FUNCTION_BLOCK TwoStateCtrl (* Template for a simple Basic Function Block Type *)
  (* Standard: 61499-2 *)
  (* Version 0.0, 2016-05-26, 4DIAC-IDE, 4DIAC *)
  (* Version 1.0, 2016-05-26, AZ, 4DIAC *)
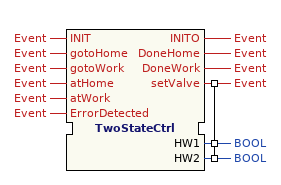
  EVENT_INPUT
    INIT; (* Initialization Request *)
    gotoHome;
    gotoWork;
    atHome;
    atWork;
    ErrorDetected;
  END_EVENT
  EVENT_OUTPUT
    INITO; (* Initialization Confirm *)
    DoneHome;
    DoneWork;
    setValve WITH HW1, HW2;
  END_EVENT
  VAR_OUTPUT
    HW1 : BOOL;
    HW2 : BOOL;
  END_VAR
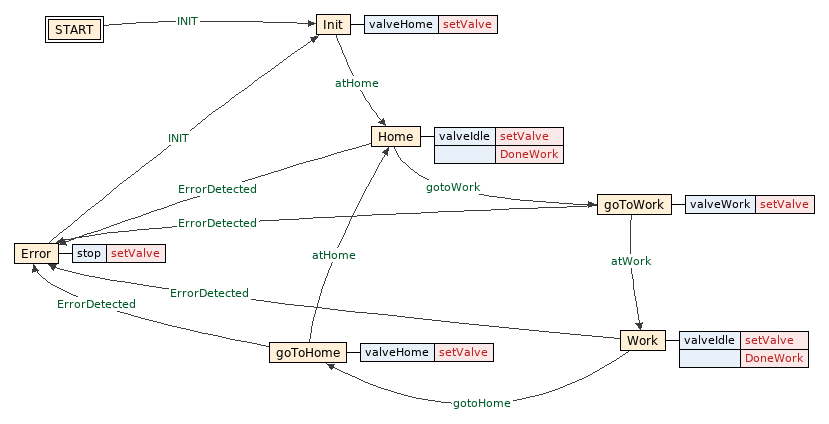
  EC_STATES
    START; (* Initial State *)
    Init : valveHome -> setValve;
    Home : valveIdle -> setValve, -> DoneWork;
    Work : valveIdle -> setValve, -> DoneWork;
    goToHome : valveHome -> setValve;
    goToWork : valveWork -> setValve;
    Error : stop -> setValve;
  END_STATES
  EC_TRANSITIONS
    START TO Init := INIT;
    Init TO Home := atHome;
    Home TO goToWork := gotoWork;
    goToWork TO Work := atWork;
    Work TO goToHome := gotoHome;
    goToHome TO Home := atHome;
    goToHome TO Error := ErrorDetected;
    Home TO Error := ErrorDetected;
    goToWork TO Error := ErrorDetected;
    Work TO Error := ErrorDetected;
    Error TO Init := INIT;
  END_TRANSITIONS
  ALGORITHM valveHome IN ST:
HW1 := true;
HW2 := false;
  END_ALGORITHM
  ALGORITHM valveWork IN ST:
HW1 := false;
HW2 := true;
  END_ALGORITHM
  ALGORITHM valveIdle IN ST:
HW1 := false;
HW2 := false;
  END_ALGORITHM
  ALGORITHM stop IN ST:
HW1 := false;
HW2 := false;
  END_ALGORITHM
END_FUNCTION_BLOCK
